(* PLC project LD_EVOLUTION_3, Beckhoff Automation GmbH TwinCAT PLC Control 3.5.10.30 *)
(* stored: creationDateTime 2019-09-26T16:15:10.9409839, modificationDateTime 2019-09-26T16:15:10.9409839 *)

PROGRAM Main
VAR
	A: BOOL;
	B: BOOL;
	Open: BOOL;
	C: BOOL;
END_VAR

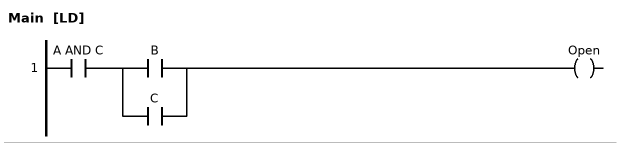
(* LD diagram, written out as Structured Text *)

Open := (A AND C) AND (B OR C);
END_PROGRAM

CONFIGURATION Application
  RESOURCE LD_EVOLUTION_3 ON PLC
    TASK PlcTask(INTERVAL := T#0ms, PRIORITY := 20);
    PROGRAM Main WITH PlcTask : Main;
  END_RESOURCE
END_CONFIGURATION
